PROGRAM MAIN
VAR
	bActivateMotion:BOOL;		//receive from ROS    sends start and stop signal
	bAuto : BOOL;				//receive from ROS    is true if we want auto mode
	bManual : BOOL;				//receive from ROS    is true if we want manual mode
	fBoomAngleRef:LREAL;			//receive from ROS	  is the desired position for the angle of the boom
	
	fPrPist : LREAL;			//sent to ROS - pressure in piston side
	fPrRod : LREAL;				//sent to ROS - pressure in rod side
	fBoomAngle:LREAL;			//sent to ROS - is the actual boom angle while crane is moving

END_VAR

P_Commissioning();
P_ControlBox();
P_CraneControl();

//SENDING TO ROS
fPrPist := G_Simulator.fPistonSidePressure;
fPrRod := G_Simulator.fRodSidePressure;
fBoomAngle := -1 * G_Simulator.fBoomAngle;


//RECEIVING FROM ROS



	
// start or stop system (through HMI buttons)
IF bActivateMotion THEN
	G_Work.bStartButton := TRUE;   //or G_Simulator.bSimulatorOn := bActivateMotion;
//ELSE
	//G_Work.bStopButton 	:= TRUE;
END_IF 

//auto or manual selection (through HMI variables)
IF bAuto THEN
	G_VirtualControlBox.bAutoSelector := FALSE;
	// set reference position
	G_VirtualControlBox.fJoystickY	:= 1 * fBoomAngleRef;				//OROR    fBoomAnimation 		: LREAL;	OR //	fBoomAngleDeg 		: LREAL;

END_IF
	
IF bManual THEN 
	G_VirtualControlBox.bAutoSelector := FALSE;
END_IF

END_PROGRAM

(* stored: Version 1.1.0.1, ProductVersion 3.1.4024.12
   POU MAIN: Id {710c49b1-6c28-4dfa-b3ee-ba840c2a49f8}, SpecialFunc None *)
